// Common 255-character string alias.
TYPE Str : STRING(255); END_TYPE

(* stored: Version 1.1.0.1
   DUT Str: Id {65794951-f31f-4956-9d1b-2c87418dbbb5} *)
